Staubli VAL3: RobotState.pjx

--- RobotState.pjx ---
Parameters version=s7.7.2 stackSize=5000 millimeterUnit=true
Program file=start.pgx
Program file=stop.pgx
Data file=RobotState.dtx

--- RobotState.dtx ---
public bool bIsValid = false
public num nRobotMode
public num nRobotStatus
public num nControlMode
public num nSequenceDelay
public bool bDrivePowered
public bool bBrakeReleased
public bool bMotionPossible
public bool bInMotion
public bool bInError
public bool bWaitAck
public bool bEStopped
public bool bValidPosition
public bool bValidVelocity
public bool bValidTorque
public bool bValidFtSensor
public bool bValidDigitalInputs
public bool bValidAnalogInputs
public jointRx jointPositions
public jointRx jointVelocities
public jointRx jointTorques
public num nFtSensorValues[6]
public bool nDigitalInputs[16]
public num nAnalogInputs[4]
